{attribute 'linkalways'}
{attribute 'hide_all_locals'}
FUNCTION_BLOCK ValueInt EXTENDS ValueIntRead IMPLEMENTS Value
VAR
END_VAR

METHOD SetFromType : BOOL
VAR_INPUT
	source : __SYSTEM.AnyType;
END_VAR
SetFromType := ConvertAnyType(source, thisAnyType);
END_METHOD

METHOD SetFromString : BOOL
VAR_INPUT
	value : T_MaxString;
END_VAR
thisValue := STRING_TO_INT(value);

SetFromString := TRUE;
END_METHOD

METHOD Set : BOOL
VAR_INPUT
	source : ANY;
END_VAR
Set := ConvertAnyType(source, thisAnyType);
END_METHOD

END_FUNCTION_BLOCK

(* stored: Version 1.1.0.1
   POU ValueInt: Id {e8f65f0d-1508-4b63-bd43-72840f736a64}, SpecialFunc None
   Method SetFromType: Id {66ed817f-e6b5-453f-a042-19ecb1c94e31}
   Method SetFromString: Id {60c24c5a-7cc7-46e7-80e8-0d7954999450}
   Method Set: Id {19961a8b-e663-49e9-ac39-11ebc7892f1a} *)
